TYPE "Type_Axis"
VERSION : 0.1
   STRUCT
      prev_pos : Real;
      prev_vel : Real;
      curr_velist : Real;
      prev_velist : Real;
      velavg_buf : Array[0.."MAX_DT"] of Real;
      dsavg_buf : Array[0.."MAX_DT"] of Real;
      dsmsavg_buf : Array[0.."MAX_DT"] of Real;
      slave : Int;
      mov_debug : Int;
      ds : Real;
      ds_ms : Real;
      stop : Bool;
      stopping : Bool;
      started : Bool;
      timeout_enabled : Bool;
      t_start : Time;
      delta_t_start : Real;
      t_mov : Time;
      delta_t_mov : Real;
      curr_timeout : Int;
      slewrate_s_up : Real;
      slewrate_s_down : Real;
      val_input : Real;
      val_input_prev : Real;
      val_output : Real;
      val_output_prev : Real;
      pid_timer {InstructionName := 'TON_TIME'; LibVersion := '1.0'} : TON_TIME;
      stat_sp_pos : Real;
      stat_sp_vel : Real;
      stat_sp_delta : Real;
      stat_sp_enable : Bool;
      stat_sp_intmode : Int;
      sp_pos : Real;
      prev_sp_pos : Real;
      sp_vel : Real;
      sp_vel_prev : Real;
      sp_delta : Real;
      sp_enable : Bool;
      interp_vmaster : Real;
      interp_vslave : Real;
      interp_dsmaster : Real;
      interp_dsslave : Real;
      interp_tmaster : Real;
      interp_tslave : Real;
      interp_rmaster : Real;
      interp_rslave : Real;
   END_STRUCT;

END_TYPE

